ABB RAPID module: PointDesignationR.mod

MODULE PointDesignationR

    CONST robtarget CameraHome:=[[337.1108,-127.6151,556.8743],[0.2459916,-0.1669462,-0.7414577,-0.601546],[1,0,1,4],[-163.8462,9E+09,9E+09,9E+09,9E+09,9E+09]];
    CONST robtarget CameraCapture:=[[239.1137,358.6136,539.5127],[0.0857302,0.05589002,-0.9655566,-0.2392219],[1,-1,1,0],[-145.4031,9E+09,9E+09,9E+09,9E+09,9E+09]];
    CONST robtarget start:=[[642.9492,-111.2745,468.2284],[0.1105639,0.6696309,0.7196313,0.1466322],[0,0,1,4],[114.9814,9E+09,9E+09,9E+09,9E+09,9E+09]];
    CONST robtarget p1:=[[563.1667,1.634485,471.787],[0.03260814,0.4073159,0.8776615,0.250481],[0,0,1,4],[147.4612,9E+09,9E+09,9E+09,9E+09,9E+09]];
    CONST robtarget p2:=[[460.5015,84.74587,473.8824],[0.008372958,-0.2721901,-0.9279103,-0.2546074],[0,0,1,4],[155.3859,9E+09,9E+09,9E+09,9E+09,9E+09]];

    CONST robtarget HomeTest:=[[332.0402,-329.8491,328.352],[0.4885546,-0.5209683,0.4893349,-0.5004576],[0,-3,1,4],[168.771,9E+09,9E+09,9E+09,9E+09,9E+09]];
    CONST robtarget HoToDis:=[[494.5024,-289.6072,161.4639],[0.01505137,-0.03083308,0.6936113,-0.7195319],[1,-1,1,4],[138.7453,9E+09,9E+09,9E+09,9E+09,9E+09]];
    CONST robtarget DisP:=[[482.48,-440.14,154.17],[0.00187341,-0.00189956,-0.707702,0.706506],[1,-2,1,4],[169.021,9E+09,9E+09,9E+09,9E+09,9E+09]];
    CONST robtarget DisPClose:=[[482.48,-378.29,154.17],[0.00187371,-0.00189861,-0.707701,0.706507],[1,-2,1,4],[169.021,9E+09,9E+09,9E+09,9E+09,9E+09]];
    CONST robtarget DisPAbove:=[[479.74,-441.56,285.22],[0.00187343,-0.00192305,-0.70768,0.706528],[1,-2,0,4],[169.013,9E+09,9E+09,9E+09,9E+09,9E+09]];
    CONST robtarget Noz1Above:=[[376.7062,-377.0453,343.9259],[0.0008304672,-0.002048479,-0.7044001,0.7097998],[0,-1,1,4],[134.22,9E+09,9E+09,9E+09,9E+09,9E+09]];
    CONST robtarget Noz1SLAbove:=[[376.7062,-377.0453,300.9713],[0.0008473364,-0.00203507,-0.7044098,0.7097901],[0,-1,1,4],[134.2202,9E+09,9E+09,9E+09,9E+09,9E+09]];
    CONST robtarget Noz1:=[[376.7062,-377.0453,279.41],[0.000817602,-0.00204644,-0.704387,0.709812],[0,-1,1,4],[134.215,9E+09,9E+09,9E+09,9E+09,9E+09]];
    CONST robtarget NozHome:=[[423.2646,-445.0486,381.9582],[0.001873649,-0.00192683,-0.7076838,0.7065242],[0,-2,0,4],[169.0306,9E+09,9E+09,9E+09,9E+09,9E+09]];
    CONST robtarget Pos_1:=[[434.8479,154.5885,276.2301],[0.2389856,-0.6773704,0.6690471,-0.1908697],[0,-1,0,0],[137.3644,9E+09,9E+09,9E+09,9E+09,9E+09]];
    CONST robtarget Pos_2:=[[508.7112,154.7467,276.2278],[0.2344545,-0.6661509,0.682647,-0.1877956],[0,-1,0,0],[137.3715,9E+09,9E+09,9E+09,9E+09,9E+09]];
    CONST robtarget Pos_3:=[[445.0982,69.16022,245.3284],[0.2387831,-0.6774528,0.6691095,-0.1906116],[2,-1,0,0],[129.9543,9E+09,9E+09,9E+09,9E+09,9E+09]];
    CONST robtarget Pos_4:=[[516.8707,70.48975,247.9003],[0.2388017,-0.6774072,0.6691476,-0.1906166],[1,-1,0,0],[130.6205,9E+09,9E+09,9E+09,9E+09,9E+09]];

    ! Camera Position for "Jars Detection" task ______ Second Approach which uses four 20 images.
    CONST robtarget Jar_1:=[[578.2363,7.590059,160.1349],[0.00247561,-0.002194457,-0.9999697,0.007042186],[1,-1,1,4],[150.582,9E+09,9E+09,9E+09,9E+09,9E+09]];
    CONST robtarget Jar_2:=[[539.0679,6.224404,160.1209],[0.002502124,-0.002170651,-0.9999694,0.007081738],[1,-1,1,4],[150.5774,9E+09,9E+09,9E+09,9E+09,9E+09]];
    CONST robtarget Jar_3:=[[506.3916,5.240112,160.1278],[0.002490915,-0.002187095,-0.9999695,0.007065233],[1,-1,1,4],[150.5787,9E+09,9E+09,9E+09,9E+09,9E+09]];
    CONST robtarget Jar_4:=[[468.2724,2.693415,160.1224],[0.002499672,-0.002171816,-0.9999694,0.007090984],[1,-1,1,4],[150.5718,9E+09,9E+09,9E+09,9E+09,9E+09]];

    CONST robtarget Jar_5:=[[467.2797,41.21567,160.1208],[0.002500687,-0.002172773,-0.9999694,0.007089187],[1,-1,1,4],[150.5729,9E+09,9E+09,9E+09,9E+09,9E+09]];
    CONST robtarget Jar_6:=[[506.2797,41.21567,160.1208],[0.002500687,-0.002172773,-0.9999694,0.007089187],[1,-1,1,4],[150.5729,9E+09,9E+09,9E+09,9E+09,9E+09]];
    CONST robtarget Jar_7:=[[539.9217,41.20918,160.1126],[0.002508863,-0.002156894,-0.9999692,0.007110072],[1,-1,1,4],[150.5725,9E+09,9E+09,9E+09,9E+09,9E+09]];
    CONST robtarget Jar_8:=[[576.3671,42.17863,160.1143],[0.002505445,-0.002157182,-0.9999692,0.007107901],[2,-1,1,4],[150.5726,9E+09,9E+09,9E+09,9E+09,9E+09]];

    CONST robtarget Jar_9:=[[575.3677,80.37881,160.1074],[0.002512477,-0.002141175,-0.9999691,0.007129352],[2,-1,1,4],[150.5705,9E+09,9E+09,9E+09,9E+09,9E+09]];
    CONST robtarget Jar_10:=[[537.2748,79.86346,160.1057],[0.002512157,-0.002139989,-0.9999691,0.007129905],[2,-1,1,4],[150.5698,9E+09,9E+09,9E+09,9E+09,9E+09]];
    CONST robtarget Jar_11:=[[502.0086,79.85998,160.1044],[0.002512725,-0.002138408,-0.9999691,0.007133875],[2,-1,1,4],[150.5689,9E+09,9E+09,9E+09,9E+09,9E+09]];
    CONST robtarget Jar_12:=[[465.7693,79.86839,160.1122],[0.002507596,-0.002156454,-0.9999692,0.007112307],[1,-1,1,4],[150.5707,9E+09,9E+09,9E+09,9E+09,9E+09]];

    CONST robtarget Jar_13:=[[465.7563,116.1511,160.1053],[0.002510817,-0.002138373,-0.9999691,0.007132343],[2,-1,1,4],[150.5686,9E+09,9E+09,9E+09,9E+09,9E+09]];
    CONST robtarget Jar_14:=[[503.1006,115.7448,160.1056],[0.0025115,-0.002136815,-0.9999691,0.007130477],[2,-1,1,4],[150.5686,9E+09,9E+09,9E+09,9E+09,9E+09]];
    CONST robtarget Jar_15:=[[538.757,114.4573,160.1061],[0.002512425,-0.002140413,-0.9999691,0.007129679],[2,-1,1,4],[150.5667,9E+09,9E+09,9E+09,9E+09,9E+09]];
    CONST robtarget Jar_16:=[[575.1255,119.2972,160.1087],[0.002503666,-0.002141883,-0.9999692,0.00712968],[2,-1,1,4],[172.0746,9E+09,9E+09,9E+09,9E+09,9E+09]];

    CONST robtarget Jar_17:=[[575.1255,155.2972,160.1087],[0.002503666,-0.002141883,-0.9999692,0.00712968],[2,-1,1,4],[172.0746,9E+09,9E+09,9E+09,9E+09,9E+09]];
    CONST robtarget Jar_18:=[[535.7615,155.2903,160.1051],[0.002497926,-0.002126256,-0.9999691,0.007146096],[2,-1,1,4],[172.0736,9E+09,9E+09,9E+09,9E+09,9E+09]];
    CONST robtarget Jar_19:=[[500.0606,153.9737,160.1045],[0.002496237,-0.002126232,-0.9999691,0.00714566],[2,-1,1,4],[172.0735,9E+09,9E+09,9E+09,9E+09,9E+09]];
    CONST robtarget Jar_20:=[[464.1317,153.2113,160.1024],[0.002497274,-0.002126625,-0.9999691,0.007149545],[2,-1,1,4],[172.0739,9E+09,9E+09,9E+09,9E+09,9E+09]];
    CONST robtarget Middle:=[[554.137,62.09487,240.156],[0.01853917,0.02127909,-0.9995263,0.01227708],[1,-1,1,4],[166.9007,9E+09,9E+09,9E+09,9E+09,9E+09]];
     ! Camera Position for "Jars Detection" task ______ First Approach which uses four images.
    VAR   robtarget Temp := [[464.1317,153.2113,160.1024],[0.002497274,-0.002126625,-0.9999691,0.007149545],[2,-1,1,4],[172.0739,9E+09,9E+09,9E+09,9E+09,9E+09]];

    CONST robtarget G{20} := [Jar_1, Jar_2, Jar_3, Jar_4, Jar_5, Jar_6, Jar_7, Jar_8, Jar_9, Jar_10, Jar_11, Jar_12, Jar_13, Jar_14, Jar_15,
        Jar_16, Jar_17, Jar_18, Jar_19, Jar_20];
    VAR num JarOnPlace{20} := [0, 0, 0, 0, 0, 0, 0, 0, 0, 0, 0, 0, 0, 0, 0, 0, 0, 0, 0, 0];
    CONST robtarget JarInPosition:=[[557.7031,199.0231,276.2335],[0.2389639,-0.6773693,0.6690513,-0.1908857],[0,-1,0,0],[137.3665,9E+09,9E+09,9E+09,9E+09,9E+09]];
    CONST robtarget JarNotInPosition:=[[557.7601,86.44871,276.2976],[0.2389937,-0.6772945,0.6690975,-0.1909521],[1,-1,0,0],[136.7944,9E+09,9E+09,9E+09,9E+09,9E+09]];

    !Nozzle positions
    VAR robtarget FirstOneOriginal:=[[364.5634,-484.9848,317.05],[0.5102121,-0.5058356,0.4925829,-0.4910968],[0,1,1,4],[146.1654,9E+09,9E+09,9E+09,9E+09,9E+09]];
    !VAR robtarget FirstOneOriginal:=[[356.2589,-488.2664,316.8112],[0.5258595,-0.4958052,0.4774238,-0.4997154],[0,-3,1,4],[-175.2839,9E+09,9E+09,9E+09,9E+09,9E+09]];
    !VAR robtarget FirstOneOriginal:=[[356.2531,-488.2716,316.8204],[0.5258421,-0.4958193,0.4774157,-0.4997275],[0,-3,1,4],[151.4595,9E+09,9E+09,9E+09,9E+09,9E+09]];
    !VAR robtarget FirstOneOriginal:=[[366.4796,-487.7165,320.9377],[0.4915279,-0.5023509,0.505054,-0.5009635],[0,1,1,4],[130.2164,9E+09,9E+09,9E+09,9E+09,9E+09]];
    VAR robtarget FirstOne:=[[356.2531,-488.2716,316.8204],[0.5258421,-0.4958193,0.4774157,-0.4997275],[0,-3,1,4],[151.4595,9E+09,9E+09,9E+09,9E+09,9E+09]];
    VAR robtarget FirstOne_20:=[[346.0473,-426.0112,432.1689],[0.5101828,-0.5058254,0.4925885,-0.4911321],[0,1,1,4],[141.0746,9E+09,9E+09,9E+09,9E+09,9E+09]];
    VAR robtarget FirstOne_21:=[[346.0473,-426.0112,432.1689],[0.5101828,-0.5058254,0.4925885,-0.4911321],[0,1,1,4],[141.0746,9E+09,9E+09,9E+09,9E+09,9E+09]];
    VAR robtarget FirstOne_13:=[[366.0591,-446.0087,432.179],[0.5101995,-0.5058179,0.4925985,-0.4911124],[0,1,1,4],[133.7709,9E+09,9E+09,9E+09,9E+09,9E+09]];
    VAR robtarget FirstOne_14:=[[346.0348,-446.0507,431.6447],[0.5101639,-0.505727,0.4926802,-0.4911611],[0,1,1,4],[148.105,9E+09,9E+09,9E+09,9E+09,9E+09]];
    VAR robtarget FirstOne_19:=[[366.0581,-426.0146,433.7001],[0.5101944,-0.5057982,0.4926129,-0.4911236],[0,1,1,4],[137.0026,9E+09,9E+09,9E+09,9E+09,9E+09]];
    VAR robtarget FirstOne_18:=[[266.2643,-445.9307,464.5445],[0.5104685,-0.5057837,0.4925609,-0.4909059],[0,1,1,4],[-118.3564,9E+09,9E+09,9E+09,9E+09,9E+09]];
    VAR robtarget FirstOne_5:=[[284.8518,-485.0245,436.239],[0.5115612,-0.5047849,0.4925893,-0.4907679],[0,1,1,4],[162.2127,9E+09,9E+09,9E+09,9E+09,9E+09]];
    VAR robtarget FirstOne_11:=[[285.39,-464.6693,439.2722],[0.5165449,-0.5008299,0.4851822,-0.4969396],[0,1,1,4],[168.0746,9E+09,9E+09,9E+09,9E+09,9E+09]];
    !opening jar lid with the right hand
    !VAR robtarget OpenJarLid_right1:=[[436.7945,-71.18093,415.3521],[0.003124756,0.7087327,0.705469,0.001334163],[0,-1,2,4],[166.2375,9E+09,9E+09,9E+09,9E+09,9E+09]];
    VAR robtarget OpenJarLid_right1:=[[436.7945,-71.18093,415.3521],[0.003124756,0.7087327,0.705469,0.001334163],[0,-1,2,4],[166.2375,9E+09,9E+09,9E+09,9E+09,9E+09]];
    VAR robtarget OpenJarLid_right1temp:=[[436.7945,-71.18093,422.3521],[0.003124756,0.7087327,0.705469,0.001334163],[0,-1,2,4],[166.2375,9E+09,9E+09,9E+09,9E+09,9E+09]];
    VAR robtarget temppp:=[[436.7945,-71.18093,421.3521],[0.003124756,0.7087327,0.705469,0.001334163],[0,-1,2,4],[166.2375,9E+09,9E+09,9E+09,9E+09,9E+09]];
    VAR jointtarget OpenJarLid_right2 := [[33.0738,-40.319,34.7805,-60.3478,90.4867,85.3075],[3.62614,9E+09,9E+09,9E+09,9E+09,9E+09]];
    VAR jointtarget OpenJarLid_right3 := [[33.0794,-39.967,34.5252,-60.3689,90.4027,14.3972],[3.62142,9E+09,9E+09,9E+09,9E+09,9E+09]];
    !points for TakeOutJarLidAndCloseJar
    VAR robtarget TakeOutJarLidAndCloseJar1:=[[548.4954,-84.25315,36.47867],[0.001396735,-0.7047526,-0.7094415,0.003806988],[1,-1,2,4],[152.5241,9E+09,9E+09,9E+09,9E+09,9E+09]];
    VAR robtarget TakeOutJarLidAndCloseJar1Temp:=[[548.4954,-84.25315,36.47867],[0.001396735,-0.7047526,-0.7094415,0.003806988],[1,-1,2,4],[152.5241,9E+09,9E+09,9E+09,9E+09,9E+09]];
    VAR robtarget TakeOutJarLidAndCloseJar2:=[[549.129,-86.93868,70.51934],[0.005022825,0.7009446,0.7131749,-0.005741474],[1,-1,2,4],[148.9269,9E+09,9E+09,9E+09,9E+09,9E+09]];
    VAR robtarget TakeOutJarLidAndCloseJar3:=[[530.686,-275.6855,198.1201],[0.005085662,0.7029518,0.7111219,0.01177542],[0,-1,1,4],[144.7235,9E+09,9E+09,9E+09,9E+09,9E+09]];
    VAR robtarget TakeOutJarLidAndCloseJar4:=[[442.0807,-71.82523,457.5505],[0.004448493,-0.7243365,-0.6894255,-0.003039069],[0,-1,2,4],[175.2385,9E+09,9E+09,9E+09,9E+09,9E+09]];
    VAR robtarget TakeOutJarLidAndCloseJar5:=[[544.5369,-219.8828,495.8261],[0.03485789,0.6806227,0.731776,0.00644785],[0,-1,1,4],[165.815,9E+09,9E+09,9E+09,9E+09,9E+09]];
    !points for closing jar lid
    VAR robtarget CloseJarLid_right1:=[[436.7945,-71.18093,415.3521],[0.003124756,0.7087327,0.705469,0.001334163],[0,-1,2,4],[166.2375,9E+09,9E+09,9E+09,9E+09,9E+09]];
    VAR jointtarget CloseJarLid_right2 := [[33.0738,-40.319,34.7805,-60.3478,90.4867,85.3075],[3.62614,9E+09,9E+09,9E+09,9E+09,9E+09]];
    VAR jointtarget CloseJarLid_right3 := [[33.0738,-40.319,34.7805,-60.3478,90.4867,85.3075],[3.62614,9E+09,9E+09,9E+09,9E+09,9E+09]];

    ! Some points to calibrate the lid on the yellow station.
    VAR robtarget Calibration_1 := [[580.5686,-88.29684,34.52171],[0.001399272,-0.7047435,-0.7094505,0.003823198],[1,-1,1,4],[152.5257,9E+09,9E+09,9E+09,9E+09,9E+09]];
    VAR robtarget Calibration_2 := [[565.8522,-88.29948,34.51547],[0.001400438,-0.7047327,-0.7094612,0.003840852],[1,-1,1,4],[152.5268,9E+09,9E+09,9E+09,9E+09,9E+09]];
    VAR robtarget Calibration_3 := [[580.5543,-88.29913,63.13507],[0.001398228,-0.7047324,-0.7094615,0.003841279],[1,-1,1,4],[152.5264,9E+09,9E+09,9E+09,9E+09,9E+09]];

    ! Points to Pick the Pippete by the right arm
    VAR robtarget PickPippete1 := [[195.649,-319.5563,313.2436],[0.7112405,-0.6988382,-0.01608902,0.07418307],[0,0,1,4],[149.918,9E+09,9E+09,9E+09,9E+09,9E+09]];
    VAR robtarget PickPippete2 := [[170.5461,-230.7654,213.2043],[0.7046992,-0.7058032,-0.01402912,0.07102092],[0,0,1,4],[157.0625,9E+09,9E+09,9E+09,9E+09,9E+09]];
    VAR robtarget PickPippete3 := [[175.5379,-131.7484,179.4989],[0.7079524,-0.7062595,0.000795693,-0.0004416163],[1,0,1,4],[156.2807,9E+09,9E+09,9E+09,9E+09,9E+09]];
    VAR robtarget PickPippeteNearPippete := [[177.2253,-197.436,179.0786],[0.7079537,-0.7062583,0.0007935975,-0.0004423254],[1,0,1,4],[156.2809,9E+09,9E+09,9E+09,9E+09,9E+09]];
    VAR robtarget PickPippeteAroundPippete := [[177.222,-131.1301,179.0808],[0.7079551,-0.7062569,0.0007965097,-0.0004404763],[1,0,1,4],[156.2794,9E+09,9E+09,9E+09,9E+09,9E+09]];
    VAR robtarget PickPippeteAroundPippeteTemp := [[175.5381,-135.7663,177.2376],[0.7079375,-0.7062744,0.0007983644,-0.0004442568],[1,0,1,4],[156.2761,9E+09,9E+09,9E+09,9E+09,9E+09]];
    VAR robtarget PickPippete4 := [[175.5398,-131.7487,239.373],[0.7079531,-0.7062589,0.0007958095,-0.0004424199],[0,0,1,4],[156.2839,9E+09,9E+09,9E+09,9E+09,9E+09]];
    VAR robtarget PickPippete9 := [[58.00851,-512.0497,345.0829],[0.4806274,-0.1937006,-0.4309853,0.7387348],[0,-1,1,4],[143.3251,9E+09,9E+09,9E+09,9E+09,9E+09]];

    VAR robtarget PickPippete4_1 := [[175.5398,-131.7487,239.373],[0.7079531,-0.7062589,0.0007958095,-0.0004424199],[0,0,1,4],[156.2839,9E+09,9E+09,9E+09,9E+09,9E+09]];
    VAR robtarget PickPippete4_2 := [[177.189,-129.7891,184.7826],[0.7079679,-0.7062441,0.0007926978,-0.0004394072],[1,0,1,4],[156.297,9E+09,9E+09,9E+09,9E+09,9E+09]];
    VAR robtarget PickPippete4_3 := [[177.1892,-131.3987,179.9682],[0.7079687,-0.7062433,0.0007927868,-0.0004407596],[1,0,1,4],[156.2953,9E+09,9E+09,9E+09,9E+09,9E+09]];
    VAR robtarget PickPippete5 := [[175.54,-84.27259,239.3745],[0.7079518,-0.7062601,0.0007943012,-0.0004460925],[0,0,1,4],[156.2846,9E+09,9E+09,9E+09,9E+09,9E+09]];
    VAR robtarget PickPippete6 := [[210.1792,-67.51133,340.1431],[0.707966,-0.7062459,0.000791344,-0.0005087436],[0,0,1,4],[156.2923,9E+09,9E+09,9E+09,9E+09,9E+09]];
    VAR robtarget PickPippete7 := [[210.188,-262.3564,340.1374],[0.7079696,-0.7062423,0.0007848368,-0.0005118064],[0,0,1,4],[156.2934,9E+09,9E+09,9E+09,9E+09,9E+09]];
    VAR robtarget PickPippete8 := [[125.4009,-534.7796,414.5038],[0.131219,-0.2493133,-0.5331899,0.7977049],[0,-2,1,4],[151.5354,9E+09,9E+09,9E+09,9E+09,9E+09]];
    !VAR robtarget PickPippete9 := [[210.188,-262.3564,340.1374],[0.7079696,-0.7062423,0.0007848368,-0.0005118064],[0,0,1,4],[156.2934,9E+09,9E+09,9E+09,9E+09,9E+09]];

    ! Points to fill in thpippetee pippete:
    VAR robtarget FillPippete1 := [[341.6258,-683.9443,511.5084],[0.3637904,0.08358209,0.7211897,-0.5835717],[0,-2,1,4],[124.8139,9E+09,9E+09,9E+09,9E+09,9E+09]];
    VAR robtarget FillPippete2 := [[62.87461,-589.7764,515.0416],[0.275436,-0.4339039,-0.530328,0.6742511],[0,-1,1,4],[83.96245,9E+09,9E+09,9E+09,9E+09,9E+09]];
    VAR robtarget FillPippete3 := [[94.98569,-349.8907,431.9817],[0.5727671,-0.7467703,-0.2549731,0.2219474],[0,0,1,4],[102.5853,9E+09,9E+09,9E+09,9E+09,9E+09]];
    VAR robtarget FillPippete4 := [[325.1082,-268.9037,457.7535],[0.6786064,-0.7311609,0.02967721,-0.06337433],[0,0,1,4],[119.312,9E+09,9E+09,9E+09,9E+09,9E+09]];
    VAR robtarget FillPippete5 := [[518.0054,-173.6114,458.7383],[0.6916274,-0.7042932,0.08632144,-0.1348009],[0,0,2,4],[141.7079,9E+09,9E+09,9E+09,9E+09,9E+09]];
    VAR robtarget FillPippete5_2 := [[325.9447,-448.3383,517.3318],[0.500117,-0.5342081,0.4917862,-0.4718592],[0,1,2,4],[19.87668,9E+09,9E+09,9E+09,9E+09,9E+09]];
    VAR robtarget FillPippete6 := [[406.7556,-112.5167,413.2942],[0.7238337,-0.6896673,-0.02013941,-0.004262863],[0,1,1,4],[111.738,9E+09,9E+09,9E+09,9E+09,9E+09]];
    VAR robtarget FillPippeteAbovePillar := [[382.0186,-119.6331,401.914],[0.7184521,-0.6954185,0.002709595,0.01457028],[0,1,1,4],[107.1083,9E+09,9E+09,9E+09,9E+09,9E+09]];
    VAR robtarget FillPippeteOnPillar := [[379.1049,-119.6783,294.4594],[0.7053983,-0.7086881,-0.009383416,0.009290063],[0,1,1,4],[109.6973,9E+09,9E+09,9E+09,9E+09,9E+09]];

    ! Points to fill out the pippetee pippete:
    VAR robtarget EmptyPippete1 := [[194.0893,-78.50488,327.2501],[0.7140521,-0.7000166,0.009698046,0.003494652],[0,0,2,4],[-157.3246,9E+09,9E+09,9E+09,9E+09,9E+09]];
    VAR robtarget EmptyPippete2 := [[210.188,-262.3564,340.1374],[0.7079696,-0.7062423,0.0007848368,-0.0005118064],[0,0,1,4],[156.2934,9E+09,9E+09,9E+09,9E+09,9E+09]];
    VAR robtarget EmptyPippeteAbovePillar := [[305.8019,-119.6324,415.2216],[0.7184599,-0.6954104,0.002705107,0.01457578],[0,0,1,4],[107.1128,9E+09,9E+09,9E+09,9E+09,9E+09]];
    VAR robtarget EmptyPippeteOnPillar := [[305.8099,-129.6291,343.5904],[0.7184706,-0.6953998,0.002716619,0.01455591],[0,0,1,4],[107.1226,9E+09,9E+09,9E+09,9E+09,9E+09]];

    ! points for the process "MovToDropNozzel"
    VAR robtarget MovToDropNozzel_1 := [[226.4902,-77.93933,422.6241],[0.7088562,-0.7053393,-0.002122149,-0.003846428],[0,0,2,4],[169.3425,9E+09,9E+09,9E+09,9E+09,9E+09]];
    VAR robtarget MovToDropNozzel_2 := [[214.2217,-84.88783,308.7547],[0.7059045,-0.7081568,-0.002914121,0.01429262],[0,0,2,4],[-162.09,9E+09,9E+09,9E+09,9E+09,9E+09]];
    VAR robtarget MovToDropNozzel_3 := [[235.3263,-130.4883,301.9571],[0.7004695,-0.698977,-0.09645084,0.1071022],[0,0,2,4],[-165.3392,9E+09,9E+09,9E+09,9E+09,9E+09]];
    VAR robtarget MovToDropNozzel_4 := [[238.051,-129.9063,296.7406],[0.7143627,-0.6905517,-0.07245048,0.08703598],[0,0,2,4],[-164.1591,9E+09,9E+09,9E+09,9E+09,9E+09]];

    VAR robtarget MovToDropNozzel_11 := [[255.6884,-123.6689,417.4043],[0.7184788,-0.6953905,0.002693033,0.0145991],[0,0,1,4],[107.1369,9E+09,9E+09,9E+09,9E+09,9E+09]];
    VAR robtarget MovToDropNozzel_22 := [[260.9324,-133.7218,343.3578],[0.7184805,-0.6953891,0.002707851,0.01457953],[0,0,1,4],[107.1803,9E+09,9E+09,9E+09,9E+09,9E+09]];


    !points to open held jar
    VAR robtarget Midd1:=[[516.37,-146.3473,438.789],[0.130924,-0.6841183,-0.6827902,-0.2205418],[0,0,1,4],[155.2096,9E+09,9E+09,9E+09,9E+09,9E+09]];
    VAR robtarget Midd2:=[[548.4106,-86.3063,203.8174],[0.03204845,0.7046776,0.7087683,-0.007059979],[0,-1,2,4],[126.0521,9E+09,9E+09,9E+09,9E+09,9E+09]];
    VAR robtarget Midd9:=[[533.0876,-139.4853,36.35339],[0.3614811,-0.9298749,-0.06503172,-0.02085684],[1,0,2,4],[148.8922,9E+09,9E+09,9E+09,9E+09,9E+09]];
    VAR robtarget Midd10:=[[555.2894,-147.5639,78.93652],[0.4163733,-0.9058304,-0.07784346,-0.006713092],[1,0,2,4],[147.3773,9E+09,9E+09,9E+09,9E+09,9E+09]];
    VAR robtarget Midd11:=[[552.0694,-185.2786,192.0681],[0.2910097,-0.9447768,-0.150038,-0.01409988],[1,0,2,4],[136.7552,9E+09,9E+09,9E+09,9E+09,9E+09]];
    VAR robtarget Midd12:=[[376.4778,-621.3032,351.6772],[0.2155167,0.121452,0.6633735,-0.7062135],[0,-2,1,4],[137.6339,9E+09,9E+09,9E+09,9E+09,9E+09]];
    VAR robtarget Midd13:=[[405.1425,-425.9179,278.2724],[0.06600403,-0.6850826,-0.6951225,0.2076298],[0,-1,1,4],[138.5983,9E+09,9E+09,9E+09,9E+09,9E+09]];
    VAR robtarget Midd14:=[[524.7402,-220.1512,231.3111],[0.08746707,-0.7491345,-0.6542986,-0.0551387],[0,0,1,4],[126.5334,9E+09,9E+09,9E+09,9E+09,9E+09]];
    VAR robtarget Midd15:=[[547.8265,-140.1339,118.4852],[0.001163659,-0.7173198,-0.6967209,0.005557916],[0,0,1,0],[106.4498,9E+09,9E+09,9E+09,9E+09,9E+09]];
    VAR robtarget Midd16:=[[537.3522,-140.5765,56.02523],[0.0006988946,0.7074742,0.706738,-0.001055677],[0,0,1,0],[95.53145,9E+09,9E+09,9E+09,9E+09,9E+09]];
    VAR robtarget Midd17:=[[537.3522,-140.5782,35.26651],[0.0006965169,0.7074735,0.7067387,-0.001056443],[0,0,1,0],[95.53266,9E+09,9E+09,9E+09,9E+09,9E+09]];
    VAR robtarget Midd18:=[[528.0477,-182.1228,174.811],[0.0147931,-0.7378669,-0.6738108,-0.0362289],[0,0,1,4],[110.359,9E+09,9E+09,9E+09,9E+09,9E+09]];
    VAR robtarget Midd19:=[[540.8347,-79.36512,185.1231],[0.02389621,0.6877341,0.7253837,-0.01640796],[0,-1,1,0],[121.6245,9E+09,9E+09,9E+09,9E+09,9E+09]];

    VAR robtarget Midd20:=[[524.5283,-396.8792,239.3516],[0.01855994,0.6776902,0.7351087,-0.002606999],[0,-1,1,4],[129.2266,9E+09,9E+09,9E+09,9E+09,9E+09]];
    VAR robtarget Midd21:=[[548.7518,-434.0228,175.894],[0.1244405,0.6483645,0.7493331,-0.05136107],[1,-1,1,4],[135.195,9E+09,9E+09,9E+09,9E+09,9E+09]];
    VAR robtarget Midd22:=[[519.0132,-376.5699,295.0557],[0.116374,-0.6922324,-0.6913291,-0.1712761],[0,-1,1,4],[158.3923,9E+09,9E+09,9E+09,9E+09,9E+09]];
    VAR robtarget Midd23:=[[632.9103,-23.5132,150.1017],[0.0006158123,0.04710628,0.9988896,0.0003107161],[1,-1,1,4],[175.2924,9E+09,9E+09,9E+09,9E+09,9E+09]];

    VAR robtarget Midd5:=[[535.7374,-133.5883,40.87439],[0.01621619,-0.7097876,-0.7039508,-0.01979489],[1,-1,1,4],[151.373,9E+09,9E+09,9E+09,9E+09,9E+09]];
    VAR robtarget Midd6:=[[528.7254,-168.0216,66.49234],[0.1161043,-0.7062157,-0.6848287,-0.1370725],[1,-1,1,4],[149.4186,9E+09,9E+09,9E+09,9E+09,9E+09]];
    VAR robtarget Midd7:=[[535.4856,-138.1096,66.77904],[0.3913096,-0.9191372,-0.02135808,-0.04009253],[1,0,1,4],[141.1107,9E+09,9E+09,9E+09,9E+09,9E+09]];
    VAR robtarget Midd8:=[[540.0371,-122.9395,36.96175],[0.3743683,-0.9270967,-0.01667459,0.007885762],[1,0,2,4],[148.7738,9E+09,9E+09,9E+09,9E+09,9E+09]];
    VAR robtarget HeldJar_PickCover:=[[550.4392,-88.55307,35.23132],[0.0004738881,-0.711928,-0.7022521,-0.0004824866],[1,-1,2,4],[151.1626,9E+09,9E+09,9E+09,9E+09,9E+09]];
    VAR robtarget HeldJar_PickCoverTemp:=[[550.8508,-90.06332,34.75971],[0.01568587,-0.7116391,-0.702301,0.009851178],[1,-1,2,4],[151.1403,9E+09,9E+09,9E+09,9E+09,9E+09]];
    VAR robtarget Midd3:=[[536.4565,-105.2238,209.9932],[0.0009176944,-0.6966414,-0.7165335,-0.03563081],[0,-1,1,4],[131.0546,9E+09,9E+09,9E+09,9E+09,9E+09]];
    VAR robtarget HeldJar_AboveJar:=[[541.1,-80.88705,166.6814],[0.01086609,0.6972497,0.7166983,-0.008257998],[0,0,1,0],[113.2381,9E+09,9E+09,9E+09,9E+09,9E+09]];
    VAR robtarget HeldJar_PlaceCover:=[[541.0815,-80.86801,150.2539],[0.01083725,0.6972349,0.716713,-0.008280328],[0,-1,1,0],[113.2341,9E+09,9E+09,9E+09,9E+09,9E+09]];
    VAR robtarget HeldJar_PlaceCover2:=[[467.9971,59.64725,138.2034],[0.0001647275,0.3948865,0.9187299,1.392494E-05],[1,-1,1,4],[155.6173,9E+09,9E+09,9E+09,9E+09,9E+09]];
    VAR robtarget Midd4:=[[545.335,-169.6051,166.0662],[0.007297219,0.6852906,0.7281541,-0.01073433],[1,-1,1,4],[138.3401,9E+09,9E+09,9E+09,9E+09,9E+09]];
    VAR jointtarget OpenHeldJarLid_right2 := [[122.646,-32.5409,13.8014,-101.023,71.2433,154.106],[-109.167,9E+09,9E+09,9E+09,9E+09,9E+09]];
    VAR robtarget Held_OpenJarLid_right1:=[[299.925,-104.7758,141.8612],[0.003347919,0.5523319,-0.8336176,-0.0001573839],[1,-1,0,4],[177.4993,9E+09,9E+09,9E+09,9E+09,9E+09]];
    VAR robtarget Held_OpenJarLid_right3 := [[466.0024,63.63331,142.2465],[0.0001546609,0.5512216,0.8343589,6.732765E-05],[1,-1,2,4],[155.6186,9E+09,9E+09,9E+09,9E+09,9E+09]];
    VAR robtarget Held_OpenJarLid_right1_Orig:=[[464.5274,59.26692,140.2369],[0.0001036231,-0.5265943,0.8501167,-0.0001247879],[1,-1,0,4],[155.6124,9E+09,9E+09,9E+09,9E+09,9E+09]];
    VAR robtarget Held_OpenJarLid_right3_Orig := [[466.1872,57.94262,140.2382],[0.000161748,0.5219612,0.8529692,3.900014E-05],[1,-1,2,4],[155.612,9E+09,9E+09,9E+09,9E+09,9E+09]];
    VAR robtarget Held_OpenJarLid_right11_Orig:=[[540.0129,-79.90893,145.1838],[0.0009086653,-0.04636181,0.9989234,0.001365947],[0,0,0,0],[105.7546,9E+09,9E+09,9E+09,9E+09,9E+09]];
    VAR robtarget Held_OpenJarLid_right33_Orig := [[540.1237,-80.10228,145.1842],[0.0008563087,-0.8882292,-0.4593977,-0.001396758],[0,0,2,0],[105.7547,9E+09,9E+09,9E+09,9E+09,9E+09]];
    VAR robtarget Held_OpenJarLid_right2 := [[467.3242,60.99391,142.2465],[0.0001546609,0.5512216,0.8343589,6.732765E-05],[1,-1,2,4],[155.6186,9E+09,9E+09,9E+09,9E+09,9E+09]];
    VAR jointtarget HeldJar_PlaceCoverAbs := [[119.341,-29.4085,15.7471,-99.831,65.08,129.757],[-107.428,9E+09,9E+09,9E+09,9E+09,9E+09]];
    VAR robtarget Held_PushingCover:=[[467.1174,60.89045,139.2775],[0.0001697346,0.1287424,0.9916781,1.377234E-05],[1,-1,1,4],[155.6257,9E+09,9E+09,9E+09,9E+09,9E+09]];
    VAR robtarget PushingPoint:=[[466.9691,60.80544,139.272],[0.0001234702,-0.5892357,0.8079612,-0.0001076188],[1,-1,0,4],[155.6251,9E+09,9E+09,9E+09,9E+09,9E+09]];

    VAR jointtarget Held_PushingCoverABS := [[122.099,-29.6605,14.5162,-99.2677,66.8305,97.9901],[-109.49,9E+09,9E+09,9E+09,9E+09,9E+09]];

    VAR robtarget Held_RightRest:=[[580.5162,-291.4563,179.9309],[0.007601542,0.7500571,0.6528434,0.1056029],[1,0,1,4],[123.5707,9E+09,9E+09,9E+09,9E+09,9E+09]];
    VAR jointtarget PushingPointABS := [[122.106,-29.6623,14.5238,-99.2724,66.8321,129.732],[-109.493,9E+09,9E+09,9E+09,9E+09,9E+09]];
    !Points to pick new filter
    VAR robtarget PickNewFilter1 := [[621.5493,-320.5108,393.9513],[0.7063952,-0.1006195,0.6996402,0.03721725],[0,1,2,4],[126.3033,9E+09,9E+09,9E+09,9E+09,9E+09]];
    VAR robtarget InsideFiltersContainer1 := [[624.0345,-425.5425,83.53399],[0.6080498,0.2930888,0.6843289,-0.2758049],[1,2,2,4],[-179.9588,9E+09,9E+09,9E+09,9E+09,9E+09]];
    VAR robtarget InsideFiltersContainer2 := [[627.1578,-426.0681,114.7737],[0.6080431,0.2930834,0.6843358,-0.2758084],[1,2,1,4],[-179.9476,9E+09,9E+09,9E+09,9E+09,9E+09]];
    VAR robtarget InsideFiltersContainer3 := [[627.1589,-424.3743,83.64411],[0.6080429,0.2930817,0.6843359,-0.2758102],[1,2,2,4],[-179.9422,9E+09,9E+09,9E+09,9E+09,9E+09]];
    VAR robtarget PickNewFilter3 := [[700.8572,-123.4617,503.5828],[0.6779857,-0.2063949,0.6670991,0.2295984],[0,1,2,4],[148.6769,9E+09,9E+09,9E+09,9E+09,9E+09]];
    VAR robtarget PlaceFilterOnBigJar := [[748.2884,-71.93338,425.3625],[0.7177004,-0.2530347,0.6101761,0.2203737],[1,1,2,4],[161.6583,9E+09,9E+09,9E+09,9E+09,9E+09]];
!    VAR robtarget PlaceFilterOnBigJar := [[746.3795,-64.11948,423.8503],[0.6907627,-0.2801198,0.6255661,0.230319],[1,1,2,4],[159.9187,9E+09,9E+09,9E+09,9E+09,9E+09]];
    VAR robtarget FilterAboveBigJar := [[736.3964,-58.74627,465.7315],[0.7179585,-0.3043995,0.571655,0.255122],[1,1,2,4],[164.984,9E+09,9E+09,9E+09,9E+09,9E+09]];
    VAR robtarget AboveFiltersContainer1 := [[624.0604,-425.5498,98.79743],[0.6080633,0.2930799,0.6843215,-0.2758029],[1,2,2,4],[-179.9616,9E+09,9E+09,9E+09,9E+09,9E+09]];
    VAR robtarget AboveFiltersContainer1_1 := [[594.6089,-425.1374,364.7184],[0.6710457,0.227214,0.6689132,-0.2250035],[0,2,1,4],[167.9116,9E+09,9E+09,9E+09,9E+09,9E+09]];
    VAR robtarget AboveFiltersContainer2 := [[624.0294,-425.5365,91.14505],[0.6080458,0.2930862,0.6843331,-0.2758062],[1,2,2,4],[-179.9555,9E+09,9E+09,9E+09,9E+09,9E+09]];
    VAR robtarget AboveFiltersContainer3 := [[624.0205,-437.218,91.17622],[0.6080415,0.2930878,0.6843355,-0.2758076],[1,2,2,4],[-179.9546,9E+09,9E+09,9E+09,9E+09,9E+09]];
    VAR robtarget AboveFiltersContainer4 := [[627.1556,-424.3723,122.1105],[0.6080418,0.2930837,0.6843366,-0.275809],[1,2,1,4],[-179.9405,9E+09,9E+09,9E+09,9E+09,9E+09]];
    VAR robtarget PickNewFilter6 := [[496.8484,-96.40296,487.0166],[0.1605303,-0.5834689,-0.756124,-0.2491398],[0,0,1,4],[166.8297,9E+09,9E+09,9E+09,9E+09,9E+09]];
    VAR robtarget PickNewFilter7 := [[457.8124,-35.79226,579.4077],[0.3662375,-0.4543677,-0.6626154,-0.4694262],[0,0,1,4],[166.312,9E+09,9E+09,9E+09,9E+09,9E+09]];
    VAR robtarget AbovePlate := [[624.5128,-458.676,421.1502],[0.5257624,0.4944812,0.4941018,-0.4846913],[1,-2,1,4],[165.4171,9E+09,9E+09,9E+09,9E+09,9E+09]];
    VAR robtarget AbovePlate_Suck := [[634.1646,-464.1222,378.8921],[0.512431,0.4822668,0.5282508,-0.4751677],[1,-2,1,4],[164.8169,9E+09,9E+09,9E+09,9E+09,9E+09]];

    !Points to pick and place funnel
    VAR robtarget PickAndPlaceFunnel1 := [[624.5128,-458.676,421.1502],[0.5257624,0.4944812,0.4941018,-0.4846913],[1,-2,1,4],[165.4171,9E+09,9E+09,9E+09,9E+09,9E+09]];
    VAR robtarget PickAndPlaceFunnel2 := [[574.0182,-349.3656,158.0238],[0.4653983,0.4840121,0.541185,0.5062168],[1,1,-1,4],[-175.8753,9E+09,9E+09,9E+09,9E+09,9E+09]];
    VAR robtarget PickAndPlaceFunnel3 := [[680.494,-358.076,380.4701],[0.5418031,-0.5262768,0.4639729,-0.4628298],[1,1,1,4],[172.4639,9E+09,9E+09,9E+09,9E+09,9E+09]];
    VAR robtarget PickAndPlaceFunnel4 := [[658.501,-109.3655,429.152],[0.6591876,-0.669107,0.2579699,-0.2263163],[1,1,2,4],[155.3449,9E+09,9E+09,9E+09,9E+09,9E+09]];
    VAR robtarget FunnelOnBigJar := [[667.3174,-109.5582,366.937],[0.66706,-0.6810696,0.2161981,-0.2107928],[1,1,2,4],[150.1866,9E+09,9E+09,9E+09,9E+09,9E+09]];
    VAR robtarget FunnelAboveBigJar := [[662.0784,-110.5511,435.6039],[0.6728038,-0.6753909,0.2155411,-0.2114811],[1,1,2,4],[149.9029,9E+09,9E+09,9E+09,9E+09,9E+09]];
    CONST robtarget NearFunnel := [[598.678,-340.9526,110.1934],[0.5140692,0.513207,0.4848319,0.4871237],[1,1,-1,4],[-173.0962,9E+09,9E+09,9E+09,9E+09,9E+09]];
    CONST robtarget AroundFunnel := [[668.3562,-341.1264,128.9281],[0.5249498,0.5178389,0.4850127,0.4701416],[1,1,-1,4],[-163.5817,9E+09,9E+09,9E+09,9E+09,9E+09]];
    CONST robtarget AboveFunnel := [[668.3507,-341.1494,188.751],[0.5249498,0.5178389,0.4850127,0.4701416],[1,1,-1,4],[-163.5817,9E+09,9E+09,9E+09,9E+09,9E+09]];


    ! Points On The Path From Main mid-Point to Orange station, to Pick jars from JarsCarrier
!    CONST robtarget PickThenPlaceJar_1 := [[221.6189,-630.9095,263.1391],[0.1033719,-0.7078362,-0.6792379,0.1640671],[0,-1,1,4],[176.5613,9E+09,9E+09,9E+09,9E+09,9E+09]];
!    CONST robtarget PickThenPlaceJar_2 := [[182.3394,-636.3591,157.7522],[0.09313875,-0.7021877,-0.6971769,0.1104628],[0,-1,0,4],[-155.607,9E+09,9E+09,9E+09,9E+09,9E+09]];
    CONST robtarget PickThenPlaceJar_1 := [[179.2008,-636.9895,308.1646],[0.02179927,0.6937607,0.7198534,0.005655664],[0,-1,0,4],[175.8574,9E+09,9E+09,9E+09,9E+09,9E+09]];
    CONST robtarget PickThenPlaceJar_2_1 := [[178.6717,-637.1774,158.8201],[0.01474175,-0.6937976,-0.7194098,0.02961638],[0,-1,0,4],[-136.568,9E+09,9E+09,9E+09,9E+09,9E+09]];
    CONST robtarget PickThenPlaceJar_2_2 := [[178.6752,-637.1756,163.6084],[0.02207202,0.69443,0.7192031,0.005167758],[0,-1,0,4],[-136.571,9E+09,9E+09,9E+09,9E+09,9E+09]];
    CONST robtarget PickThenPlaceJar_3 := [[514.5727,-92.31973,311.4816],[0.02578642,-0.03406016,0.9988954,-0.0195672],[0,-1,1,4],[152.8023,9E+09,9E+09,9E+09,9E+09,9E+09]];
    CONST robtarget PickThenPlaceJar_4 := [[540.8358,-79.04424,241.8575],[0.01282984,-0.01291086,0.9998207,-0.005222363],[0,-1,1,4],[140.2428,9E+09,9E+09,9E+09,9E+09,9E+09]];
    CONST robtarget PickThenPlaceJar_5 := [[540.033,-79.02003,170.1638],[0.01224879,-0.01340815,0.9998229,-0.004945346],[1,-1,1,4],[140.5999,9E+09,9E+09,9E+09,9E+09,9E+09]];
    CONST robtarget PickThenPlaceJar_4_2 := [[540.827,-21.1302,241.8817],[0.01285445,-0.01293795,0.9998198,-0.005274247],[1,-1,1,4],[140.2354,9E+09,9E+09,9E+09,9E+09,9E+09]];
    CONST robtarget PickThenPlaceJar_5_2 := [[540.8089,-21.14899,197.2088],[0.01277829,-0.01288883,0.9998217,-0.005204006],[1,-1,1,4],[140.2409,9E+09,9E+09,9E+09,9E+09,9E+09]];
    CONST robtarget PickThenPlaceJar_5_3 := [[540.8538,-45.851,197.211],[0.01278042,-0.0128894,0.9998217,-0.005203976],[1,-1,1,4],[140.2329,9E+09,9E+09,9E+09,9E+09,9E+09]];


    CONST robtarget FilterFormMissileToPlate1 := [[705.6249,-118.5424,547.73],[0.7170886,-0.1016343,0.6858905,0.07077146],[1,0,-1,5],[173.9745,9E+09,9E+09,9E+09,9E+09,9E+09]];
    CONST robtarget FilterFormMissileToPlate2 := [[753.3035,-132.1059,435.7927],[0.7123696,-0.0763738,0.6961165,0.04602613],[1,0,-1,5],[171.6446,9E+09,9E+09,9E+09,9E+09,9E+09]];
    CONST robtarget FilterFormMissileToPlate3 := [[753.3035,-139.1056,418.2421],[0.7123706,-0.07637336,0.6961155,0.04602607],[1,0,-1,5],[171.6473,9E+09,9E+09,9E+09,9E+09,9E+09]];
    CONST robtarget FilterFormMissileToPlate4 := [[753.2958,-57.30429,442.5074],[0.7123702,-0.07635287,0.6961184,0.04602309],[1,0,-1,5],[171.6511,9E+09,9E+09,9E+09,9E+09,9E+09]];
    CONST robtarget FilterFormMissileToPlate5 := [[753.2941,-57.30222,411.2484],[0.7123696,-0.07635479,0.6961186,0.04602571],[1,0,-1,5],[171.6533,9E+09,9E+09,9E+09,9E+09,9E+09]];

    !Points to push filter on big jar
    VAR robtarget PushFilter1 := [[756.0059,-13.61446,394.8519],[0.02664099,-0.762088,-0.2717999,-0.5870579],[1,0,0,5],[170.9841,9E+09,9E+09,9E+09,9E+09,9E+09]];
    VAR robtarget PushFilter2 := [[756.8353,-17.41819,380.0923],[0.02663975,-0.7620836,-0.2718007,-0.5870632],[1,0,0,5],[170.9992,9E+09,9E+09,9E+09,9E+09,9E+09]];
    VAR robtarget PushFilter3 := [[749.9757,-27.72997,380.5538],[0.02663724,-0.762088,-0.2718012,-0.5870575],[1,0,1,5],[170.9892,9E+09,9E+09,9E+09,9E+09,9E+09]];
    VAR robtarget PushFilter4 := [[743.4111,-33.86438,380.5558],[0.02663806,-0.7620863,-0.2718004,-0.5870599],[1,0,1,5],[170.9918,9E+09,9E+09,9E+09,9E+09,9E+09]];
    VAR robtarget PushFilter5 := [[737.4625,-40.36673,380.5567],[0.02663708,-0.7620859,-0.2718003,-0.5870607],[1,0,1,5],[170.9944,9E+09,9E+09,9E+09,9E+09,9E+09]];
    VAR robtarget PushFilter6 := [[733.3664,-46.5193,380.5568],[0.02663536,-0.7620849,-0.2718024,-0.587061],[1,0,1,5],[170.9958,9E+09,9E+09,9E+09,9E+09,9E+09]];
    VAR robtarget PushFilter7 := [[733.374,-46.5389,389.5945],[0.02661256,-0.7620885,-0.2717963,-0.5870603],[1,0,1,5],[170.9965,9E+09,9E+09,9E+09,9E+09,9E+09]];
    VAR robtarget PushFilter8 := [[733.368,-46.54215,458.1636],[0.02660939,-0.7620866,-0.2717976,-0.5870622],[1,1,0,5],[170.9965,9E+09,9E+09,9E+09,9E+09,9E+09]];
    VAR robtarget PushFilter9 := [[741.5504,-50.15194,502.4712],[0.1524157,0.3446489,0.7166551,0.5868492],[1,0,1,4],[175.4269,9E+09,9E+09,9E+09,9E+09,9E+09]];
    VAR robtarget PushFilter10 := [[736.2281,-82.81029,382.6262],[0.5206777,-0.2948277,0.801129,-0.01278638],[1,1,2,5],[162.8944,9E+09,9E+09,9E+09,9E+09,9E+09]];
    VAR robtarget PushFilter11 := [[724.3495,-65.00657,382.1458],[0.527997,-0.3223275,0.7825246,0.0705651],[1,1,2,5],[159.5265,9E+09,9E+09,9E+09,9E+09,9E+09]];
    VAR robtarget PushFilter12 := [[728.5455,-49.11105,419.8861],[0.5490216,-0.3086144,0.7727147,0.07902226],[1,1,2,5],[161.8061,9E+09,9E+09,9E+09,9E+09,9E+09]];
    VAR robtarget PushFilter13 := [[743.5784,25.86427,430.176],[0.6582333,-0.2462072,0.6854758,0.1903519],[1,1,2,0],[121.1031,9E+09,9E+09,9E+09,9E+09,9E+09]];
    VAR robtarget PushFilter14 := [[733.2577,-46.34735,458.0763],[0.5866504,-0.3494981,0.7297264,-0.03452196],[1,1,2,5],[170.9967,9E+09,9E+09,9E+09,9E+09,9E+09]];
    VAR robtarget PushFilter15 := [[801.3381,-85.08338,551.8134],[0.510915,0.341691,0.7031891,0.3574048],[0,0,1,0],[130.876,9E+09,9E+09,9E+09,9E+09,9E+09]];
    VAR robtarget PushFilter16 := [[664.3308,-108.3452,397.178],[0.006608484,0.4401534,0.897898,0.0006642516],[0,0,1,0],[130.8481,9E+09,9E+09,9E+09,9E+09,9E+09]];
    VAR robtarget PushFilter17 := [[664.3331,-108.3433,384.4006],[0.006609402,0.4401523,0.8978986,0.0006644762],[0,0,1,0],[130.8402,9E+09,9E+09,9E+09,9E+09,9E+09]];
    VAR robtarget PushFilter18 := [[651.4076,-117.9172,384.3516],[0.006577531,0.4400893,0.8979297,0.0006210515],[1,0,1,0],[130.8029,9E+09,9E+09,9E+09,9E+09,9E+09]];
    VAR robtarget PushFilter19 := [[733.2577,-46.34735,458.0763],[0.5866504,-0.3494981,0.7297264,-0.03452196],[1,1,2,5],[170.9967,9E+09,9E+09,9E+09,9E+09,9E+09]];
    VAR robtarget PushFilter20 := [[720.921,-63.57402,380.5577],[0.02661204,-0.762087,-0.2717952,-0.5870627],[1,0,1,5],[170.9985,9E+09,9E+09,9E+09,9E+09,9E+09]];

    !points to PutUsedFilterInPlate
    VAR robtarget PutUsedFilterInPlate1 := [[473.6227,-252.2065,279.1347],[0.6325881,-0.7069083,0.292002,-0.1218517],[1,0,2,4],[-165.909,9E+09,9E+09,9E+09,9E+09,9E+09]];
    VAR robtarget PutUsedFilterInPlate2:= [[574.4794,-235.4697,49.00514],[0.4863034,-0.4829491,0.5373127,-0.4914918],[1,1,1,4],[-157.2493,9E+09,9E+09,9E+09,9E+09,9E+09]];
    VAR robtarget PutUsedFilterInPlate3 := [[514.0889,-247.6884,143.5489],[0.4872082,-0.5422345,0.4708532,-0.4968975],[1,1,1,4],[-159.2458,9E+09,9E+09,9E+09,9E+09,9E+09]];
    VAR robtarget PutUsedFilterInPlate4 := [[530.6711,-252.6093,318.137],[0.599079,-0.5827813,0.4087358,-0.3666134],[1,1,1,4],[-160.9291,9E+09,9E+09,9E+09,9E+09,9E+09]];
    VAR robtarget PutUsedFilterInPlate5 := [[391.5533,-233.6493,580.6913],[0.7759497,-0.6290888,-0.033647,-0.03189521],[1,0,2,4],[178.5084,9E+09,9E+09,9E+09,9E+09,9E+09]];
    VAR robtarget PutUsedFilterInPlate6 := [[566.8242,-237.7017,335.2878],[0.2433534,0.3150106,0.7158626,0.5736622],[1,0,0,4],[172.7277,9E+09,9E+09,9E+09,9E+09,9E+09]];
    VAR robtarget PlateInPlace := [[627.95,-154.2937,333.2767],[0.1975931,0.2695499,0.6932085,0.6385622],[1,0,0,4],[166.0525,9E+09,9E+09,9E+09,9E+09,9E+09]];

    !Points for BorderingFilterToPutInPlate
    VAR robtarget BorderingFilterToPutInPlate1 := [[675.6477,-214.1475,507.9201],[0.004738619,-0.7108954,-0.0161659,-0.7030959],[1,-2,-1,4],[175.1633,9E+09,9E+09,9E+09,9E+09,9E+09]];
    VAR robtarget BorderingFilterToPutInPlate2 := [[113.5013,-37.46609,79.09233],[0.02876629,0.7071135,-0.03476489,0.7056588],[1,-2,0,4],[127.6906,9E+09,9E+09,9E+09,9E+09,9E+09]];
    VAR robtarget BorderingFilterToPutInPlate3 := [[93.81635,6.562484,57.52491],[0.09276452,0.6824939,0.09494647,0.7187364],[1,-2,-1,4],[127.7968,9E+09,9E+09,9E+09,9E+09,9E+09]];
    VAR robtarget BorderingFilterToPutInPlate4 := [[88.22985,31.19816,53.94881],[0.07252922,0.6804215,0.1459732,0.7144634],[1,-2,0,4],[128.4669,9E+09,9E+09,9E+09,9E+09,9E+09]];
    VAR robtarget BorderingFilterToPutInPlate5 := [[77.45119,62.40168,52.68208],[0.05411451,0.6635692,0.1976721,0.7194952],[1,-2,0,4],[129.3063,9E+09,9E+09,9E+09,9E+09,9E+09]];
    VAR robtarget BorderingFilterToPutInPlate6 := [[567.22,-173.2041,316.7787],[0.2664002,0.3040051,0.6687229,0.6240364],[1,0,0,4],[-160.9951,9E+09,9E+09,9E+09,9E+09,9E+09]];

    !Points to Move plate from stack to red piece near big jar
    VAR robtarget MovePlateFromStackToRedLocation1 := [[567.22,-173.2041,316.7787],[0.2664002,0.3040051,0.6687229,0.6240364],[1,0,0,4],[-160.9951,9E+09,9E+09,9E+09,9E+09,9E+09]];
    VAR robtarget MovePlateFromStackToRedLocation2 := [[567.22,-173.2041,316.7787],[0.2664002,0.3040051,0.6687229,0.6240364],[1,0,0,4],[-160.9951,9E+09,9E+09,9E+09,9E+09,9E+09]];
    VAR robtarget MovePlateFromStackToRedLocation3 := [[567.22,-173.2041,316.7787],[0.2664002,0.3040051,0.6687229,0.6240364],[1,0,0,4],[-160.9951,9E+09,9E+09,9E+09,9E+09,9E+09]];
    VAR robtarget MovePlateFromStackToRedLocation4 := [[567.22,-173.2041,316.7787],[0.2664002,0.3040051,0.6687229,0.6240364],[1,0,0,4],[-160.9951,9E+09,9E+09,9E+09,9E+09,9E+09]];
    VAR robtarget MovePlateFromStackToRedLocation5 := [[567.22,-173.2041,316.7787],[0.2664002,0.3040051,0.6687229,0.6240364],[1,0,0,4],[-160.9951,9E+09,9E+09,9E+09,9E+09,9E+09]];
    VAR robtarget MovePlateFromStackToRedLocation6 := [[567.22,-173.2041,316.7787],[0.2664002,0.3040051,0.6687229,0.6240364],[1,0,0,4],[-160.9951,9E+09,9E+09,9E+09,9E+09,9E+09]];
    VAR robtarget MovePlateFromStackToRedLocation7 := [[567.22,-173.2041,316.7787],[0.2664002,0.3040051,0.6687229,0.6240364],[1,0,0,4],[-160.9951,9E+09,9E+09,9E+09,9E+09,9E+09]];
    VAR robtarget MovePlateFromStackToRedLocation8 := [[567.22,-173.2041,316.7787],[0.2664002,0.3040051,0.6687229,0.6240364],[1,0,0,4],[-160.9951,9E+09,9E+09,9E+09,9E+09,9E+09]];

    ! Some points to pick the plate
    VAR robtarget PickPlate1 := [[227.1261,-527.5699,341.0041],[0.04053182,-0.8623218,-0.4814033,0.1516877],[0,-1,1,4],[176.1331,9E+09,9E+09,9E+09,9E+09,9E+09]];
    VAR robtarget PickPlate2 := [[-3.567228,-408.2107,134.7796],[0.3952619,-0.6121742,-0.4965889,0.471604],[0,-1,1,4],[-130.3624,9E+09,9E+09,9E+09,9E+09,9E+09]];
    VAR robtarget PickPlate3 := [[-142.6978,-318.9195,42.63297],[0.4808339,-0.4860117,-0.518315,0.5137518],[1,-1,1,4],[-143.24,9E+09,9E+09,9E+09,9E+09,9E+09]];
    VAR robtarget PickPlate4 := [[-142.4758,-318.8727,61.93118],[0.4808406,-0.4865499,-0.5182256,0.5133262],[1,-1,1,4],[-143.2737,9E+09,9E+09,9E+09,9E+09,9E+09]];
    VAR robtarget PickPlate5 := [[-77.97506,-326.9365,96.9474],[0.5010442,-0.5218936,-0.4985341,0.4775413],[0,-1,1,4],[-136.8395,9E+09,9E+09,9E+09,9E+09,9E+09]];
    VAR robtarget PickPlate6 := [[-90.30951,-320.5932,44.24039],[0.4979136,-0.5123259,-0.5073266,0.4818961],[1,-1,1,4],[-143.0363,9E+09,9E+09,9E+09,9E+09,9E+09]];
    VAR robtarget PickPlate7 := [[-61.84347,-321.6961,44.76805],[0.4966117,-0.5100227,-0.50834,0.4846072],[1,-1,1,4],[-142.9827,9E+09,9E+09,9E+09,9E+09,9E+09]];
    VAR robtarget PickPlate8 := [[-52.97003,-322.5573,106.2267],[0.4950693,-0.5096297,-0.5090222,0.485881],[0,-1,1,4],[-142.9297,9E+09,9E+09,9E+09,9E+09,9E+09]];
    VAR robtarget PickPlate9 := [[-44.28172,-319.6465,128.838],[0.6372106,-0.3134488,-0.6291855,-0.3159717],[0,-1,0,4],[-133.2934,9E+09,9E+09,9E+09,9E+09,9E+09]];
    VAR robtarget PickPlate10_1 := [[-143.5759,-241.5467,111.6477],[0.6093763,-0.4017231,-0.5714734,-0.3750964],[0,-1,0,4],[-141.1836,9E+09,9E+09,9E+09,9E+09,9E+09]];
    VAR robtarget PickPlate10_2 := [[-167.7915,-241.5351,118.1164],[0.6093708,-0.4017192,-0.571467,-0.3751193],[0,-1,0,4],[-141.1944,9E+09,9E+09,9E+09,9E+09,9E+09]];
    VAR robtarget PickPlate10_3 := [[-167.7915,-241.5351,123.1164],[0.6093708,-0.4017192,-0.571467,-0.3751193],[0,-1,0,4],[-141.1944,9E+09,9E+09,9E+09,9E+09,9E+09]];
    VAR robtarget PickPlate10_4 := [[-37.56079,-321.5652,103.587],[0.547386,-0.3171856,-0.6532114,-0.416025],[1,-1,0,4],[-144.1172,9E+09,9E+09,9E+09,9E+09,9E+09]];
    VAR robtarget PickPlate11_Down := [[-143.5759,-241.5467,134.8745],[0.6093763,-0.4017231,-0.5714734,-0.3750964],[0,-1,0,4],[-141.1836,9E+09,9E+09,9E+09,9E+09,9E+09]];
    VAR robtarget PickPlate11_Up := [[-143.5759,-241.5467,134.8745],[0.6093763,-0.4017231,-0.5714734,-0.3750964],[0,-1,0,4],[-141.1836,9E+09,9E+09,9E+09,9E+09,9E+09]];
    VAR robtarget PickPlate12 := [[-241.0147,-241.6081,137.761],[0.616179,-0.391013,-0.5779745,-0.3652091],[0,-1,0,4],[-141.1788,9E+09,9E+09,9E+09,9E+09,9E+09]];
    VAR robtarget PickPlate13 := [[-241.1691,-241.7823,111.6477],[0.6093817,-0.4017254,-0.5714735,-0.3750848],[1,-1,0,4],[-141.1598,9E+09,9E+09,9E+09,9E+09,9E+09]];
    VAR robtarget PickPlate14_ThrowPlateCover := [[-74.80486,-257.3926,223.272],[0.5064288,-0.4275604,-0.5680993,-0.4878372],[0,0,0,4],[-151.8755,9E+09,9E+09,9E+09,9E+09,9E+09]];

    ! Some points to put plate in Capinet

    VAR robtarget PutPlateInCapinet1PreMoving := [[622.3975,-163.4876,346.3798],[0.2100825,0.2565895,0.7139377,0.616701],[1,0,0,4],[161.9459,9E+09,9E+09,9E+09,9E+09,9E+09]];
    VAR robtarget PutPlateInCapinet1 := [[336.9954,-126.1508,641.6207],[0.2318186,0.05682539,-0.6800953,-0.6931821],[1,0,1,4],[-162.4004,9E+09,9E+09,9E+09,9E+09,9E+09]];
    VAR robtarget PutPlateInCapinet2 := [[107.7427,-67.06541,778.0781],[0.3994297,0.347616,-0.6359779,-0.5613832],[1,0,1,4],[-121.987,9E+09,9E+09,9E+09,9E+09,9E+09]];
    VAR robtarget PutPlateInCapinet3 := [[-39.04373,-73.9049,744.7962],[0.4666459,0.476293,-0.5254644,-0.5284635],[1,0,1,4],[-116.1677,9E+09,9E+09,9E+09,9E+09,9E+09]];
    VAR robtarget PutPlateInCapinet4 := [[23.16677,-73.90886,713.7164],[0.4666705,0.4762923,-0.5254518,-0.5284551],[1,0,1,4],[-116.1661,9E+09,9E+09,9E+09,9E+09,9E+09]];
    VAR robtarget PutPlateInCapinet5 := [[-39.03989,-73.90785,713.7233],[0.466655,0.476292,-0.5254535,-0.5284672],[1,0,1,4],[-116.1664,9E+09,9E+09,9E+09,9E+09,9E+09]];
    VAR robtarget PutPlateInCapinet6 := [[-37.01698,-73.91552,761.9521],[0.466686,0.4762945,-0.5254425,-0.5284486],[1,0,1,4],[-116.1639,9E+09,9E+09,9E+09,9E+09,9E+09]];
    VAR robtarget PutPlateInCapinet7 := [[-212.6318,-334.0861,481.3083],[0.6006479,-0.400857,-0.606375,-0.3329342],[0,-1,-1,4],[-113.8211,9E+09,9E+09,9E+09,9E+09,9E+09]];
    VAR robtarget PutPlateInCapinet8 := [[-212.6318,-334.0861,481.3083],[0.6006479,-0.400857,-0.606375,-0.3329342],[0,-1,-1,4],[-113.8211,9E+09,9E+09,9E+09,9E+09,9E+09]];
    VAR robtarget PutPlateInCapinet9 := [[-212.6318,-334.0861,481.3083],[0.6006479,-0.400857,-0.606375,-0.3329342],[0,-1,-1,4],[-113.8211,9E+09,9E+09,9E+09,9E+09,9E+09]];

    !points to take out the plate from the closet

    VAR robtarget AbovePlateInCloset := [[-37.01698,-73.91552,791.9521],[0.466686,0.4762945,-0.5254425,-0.5284486],[1,0,1,4],[-116.1639,9E+09,9E+09,9E+09,9E+09,9E+09]];
    VAR robtarget AroundPlateInCloset := [[-36.92104,-73.94338,713.5489],[0.466785,0.4762551,-0.5253302,-0.5285084],[1,0,1,4],[-116.1534,9E+09,9E+09,9E+09,9E+09,9E+09]];
    VAR robtarget TakePlateOut1 := [[153.3338,-128.2487,793.0741],[0.4162462,0.5471437,-0.473133,-0.5509248],[1,0,1,4],[-119.9038,9E+09,9E+09,9E+09,9E+09,9E+09]];
    VAR robtarget TakePlateOut2 := [[653.3688,-154.808,526.8815],[0.1977761,0.3044988,0.6442697,0.6731133],[1,-1,1,4],[-155.923,9E+09,9E+09,9E+09,9E+09,9E+09]];
    VAR robtarget PlateAboveBigJar := [[666.7081,-111.3742,401.4151],[0.2972408,0.3367108,0.6372746,0.6262226],[1,-1,1,4],[-165.2874,9E+09,9E+09,9E+09,9E+09,9E+09]];
    VAR robtarget PlateOnBigJar := [[666.7331,-111.2638,365.1944],[0.2982312,0.3357119,0.6368653,0.6267043],[1,-1,1,4],[-165.2628,9E+09,9E+09,9E+09,9E+09,9E+09]];
    VAR robtarget PlateOnBigJar1 := [[666.7374,-111.2572,359.6436],[0.2982137,0.3356809,0.6368814,0.6267129],[1,0,0,4],[-165.2619,9E+09,9E+09,9E+09,9E+09,9E+09]];


    !Points tp pick the filter for analysis
    VAR robtarget PickFilterForAnalysis1 := [[675.5394,-108.0748,503.7346],[0.6090953,-0.2344455,0.7329304,0.1919672],[1,-1,0,4],[-175.308,9E+09,9E+09,9E+09,9E+09,9E+09]];
    VAR robtarget AboveFilterForAnalysis := [[718.9147,-65.57491,471.2317],[0.6941316,-0.2419525,0.6493869,0.1947739],[1,-1,0,5],[170.0938,9E+09,9E+09,9E+09,9E+09,9E+09]];
    VAR robtarget PickFilterForAnalysis := [[732.3462,-74.86136,412.2591],[0.6741185,-0.220105,0.6811666,0.1820167],[1,-1,0,5],[166.8679,9E+09,9E+09,9E+09,9E+09,9E+09]];


   !poibnts to remove the plate after the analysis
    VAR robtarget MovePlateAfterAnalysis1 := [[732.3462,-74.86136,412.2591],[0.6741185,-0.220105,0.6811666,0.1820167],[1,-1,0,5],[166.8679,9E+09,9E+09,9E+09,9E+09,9E+09]];
    VAR robtarget MovePlateAfterAnalysis2 := [[732.3462,-74.86136,412.2591],[0.6741185,-0.220105,0.6811666,0.1820167],[1,-1,0,5],[166.8679,9E+09,9E+09,9E+09,9E+09,9E+09]];
    VAR robtarget MovePlateAfterAnalysis3 := [[663.5577,-116.3641,387.2455],[0.02010107,0.574471,0.818178,0.01280024],[0,-1,1,0],[140.1178,9E+09,9E+09,9E+09,9E+09,9E+09]];
    VAR robtarget MovePlateAfterAnalysis4 := [[663.5488,-116.4332,398.0156],[0.02007263,0.5745333,0.8181344,0.0128338],[0,-1,1,0],[140.1235,9E+09,9E+09,9E+09,9E+09,9E+09]];
    VAR robtarget MovePlateAfterAnalysis5 := [[462.5022,-435.4173,392.7523],[0.02093044,0.6087145,0.792644,0.02727618],[0,-1,1,4],[140.0694,9E+09,9E+09,9E+09,9E+09,9E+09]];
    VAR robtarget MovePlateAfterAnalysis6 := [[484.446,-345.5098,107.2954],[0.05076824,-0.699346,-0.7125604,-0.02440064],[1,-1,1,4],[156.0081,9E+09,9E+09,9E+09,9E+09,9E+09]];
    VAR robtarget MovePlateAfterAnalysis7 := [[462.8721,-336.8476,46.51273],[0.03607976,-0.6682198,-0.7430834,-0.002757301],[1,-1,1,4],[154.5291,9E+09,9E+09,9E+09,9E+09,9E+09]];



    !Points to CloseCapinet
    VAR robtarget CloseCapinet1 := [[207.5222,-242.1754,591.3132],[0.06543734,-0.0622346,-0.6650254,-0.7413408],[1,0,1,4],[-170.9305,9E+09,9E+09,9E+09,9E+09,9E+09]];
    VAR robtarget CloseCapinet2 := [[-22.68939,-315.5607,560.8279],[0.2878203,-0.207479,-0.611744,-0.7070227],[1,0,2,4],[102.4968,9E+09,9E+09,9E+09,9E+09,9E+09]];
    VAR robtarget CloseCapinet3 := [[-120.784,-345.9569,597.4397],[0.3498625,0.001832771,-0.5227011,-0.7774165],[1,1,2,4],[98.65139,9E+09,9E+09,9E+09,9E+09,9E+09]];
    VAR robtarget CloseCapinet4 := [[-82.97842,-382.2726,644.6324],[0.03086359,-0.1110591,0.3303497,0.9367937],[1,0,1,4],[98.49933,9E+09,9E+09,9E+09,9E+09,9E+09]];
    VAR robtarget CloseCapinet5 := [[-33.28422,-393.3404,662.8998],[0.05534496,-0.08431086,-0.2613863,-0.9599509],[1,0,1,4],[100.3842,9E+09,9E+09,9E+09,9E+09,9E+09]];
    VAR robtarget CloseCapinet6 := [[126.8073,-299.3019,691.0593],[0.1787152,-0.2536302,-0.5090077,-0.8028972],[1,0,1,4],[166.1153,9E+09,9E+09,9E+09,9E+09,9E+09]];
    VAR robtarget CloseCapinet7 := [[195.0965,-120.0588,719.5216],[0.4439963,-0.1593523,-0.7213333,-0.507102],[1,0,1,4],[-150.4515,9E+09,9E+09,9E+09,9E+09,9E+09]];
    VAR robtarget CloseCapinet8 := [[96.39011,-1.393748,742.2653],[0.5350459,-0.062455,-0.7222924,-0.4337268],[1,0,1,4],[-138.2767,9E+09,9E+09,9E+09,9E+09,9E+09]];
    VAR robtarget CloseCapinet9 := [[63.36932,10.57348,768.642],[0.6800932,-0.05562977,-0.7297705,-0.04258671],[1,0,2,4],[-133.4059,9E+09,9E+09,9E+09,9E+09,9E+09]];
    VAR robtarget CloseCapinet10 := [[52.19879,11.1265,767.5461],[0.6809717,-0.0249305,-0.7318537,-0.006795681],[1,0,1,4],[-132.5736,9E+09,9E+09,9E+09,9E+09,9E+09]];

    VAR robtarget MoveDispenser1 := [[382.0439,-119.625,292.9677],[0.7184659,-0.6954051,0.002741368,0.01452396],[0,1,1,4],[107.1018,9E+09,9E+09,9E+09,9E+09,9E+09]];
    VAR robtarget MoveDispenser2 := [[367.2742,-97.70506,472.0224],[0.7114094,-0.7025003,0.004124381,-0.0193076],[0,0,2,4],[137.8868,9E+09,9E+09,9E+09,9E+09,9E+09]];
    VAR robtarget MoveDispenser3 := [[296.933,-82.52208,478.6049],[0.7070982,-0.7064348,0.02777747,-0.01379868],[0,0,2,4],[145.1462,9E+09,9E+09,9E+09,9E+09,9E+09]];
    VAR robtarget MoveDispenser31 := [[296.933,-98.82317,447.6208],[0.705121,-0.7090259,0.003036739,-0.008797801],[0,0,2,4],[148.4961,9E+09,9E+09,9E+09,9E+09,9E+09]];
    VAR robtarget MoveDispenser4 := [[296.933,-113.715,419.1608],[0.7027627,-0.7111467,-0.01941378,-0.004263762],[0,0,2,4],[151.5516,9E+09,9E+09,9E+09,9E+09,9E+09]];
    VAR robtarget MoveDispenser5 := [[296.933,-135.4433,412.0101],[0.7132996,-0.7001655,0.0264315,-0.01653659],[0,0,1,4],[124.0881,9E+09,9E+09,9E+09,9E+09,9E+09]];
    VAR robtarget MoveDispenser6_1 := [[296.9357,-144.6807,396.5883],[0.7462527,-0.665211,0.02072768,-0.0131015],[0,0,2,4],[167.538,9E+09,9E+09,9E+09,9E+09,9E+09]];
    VAR robtarget MoveDispenser6_2 := [[296.9381,-144.6735,396.579],[0.727263,-0.685921,0.02034875,-0.01366454],[0,0,2,4],[167.5494,9E+09,9E+09,9E+09,9E+09,9E+09]];
    VAR robtarget MoveDispenser7 := [[295.9322,-206.0766,442.1875],[0.7091605,-0.7050132,0.005624216,0.004032394],[0,0,2,4],[138.4178,9E+09,9E+09,9E+09,9E+09,9E+09]];
    VAR robtarget MoveDispenser8 := [[316.067,-25.3562,539.6172],[0.5164476,-0.4981974,0.4920629,0.492905],[0,1,3,4],[114.3105,9E+09,9E+09,9E+09,9E+09,9E+09]];
    VAR robtarget MoveDispenser9 := [[324.9807,-24.98611,513.7685],[0.4891407,-0.4735606,0.5265107,0.5091838],[0,1,3,4],[118.2191,9E+09,9E+09,9E+09,9E+09,9E+09]];
    VAR robtarget MoveDispenser10 := [[325.1716,-25.00177,494.9056],[0.4893806,-0.4731246,0.5266935,0.5091697],[0,1,2,4],[113.0836,9E+09,9E+09,9E+09,9E+09,9E+09]];
    VAR robtarget MoveDispenser10Clear := [[325.1701,-25.00095,491.0015],[0.4893791,-0.4731236,0.526693,0.5091724],[0,1,2,4],[113.0846,9E+09,9E+09,9E+09,9E+09,9E+09]];
    VAR robtarget MoveDispenser11 := [[292.933,-189.7269,398.1999],[0.7107903,-0.7032589,0.01307814,0.005744404],[0,0,1,4],[140.9083,9E+09,9E+09,9E+09,9E+09,9E+09]];
    VAR robtarget MoveDispenser12 := [[296.933,-133.6059,398.1976],[0.7107857,-0.7032634,0.01308545,0.005749269],[0,0,1,4],[140.8967,9E+09,9E+09,9E+09,9E+09,9E+09]];

    ! Points to ensure Tight Equipment of the nozzle
    VAR robtarget TightEquipping_1 := [[535.3924,-105.5459,384.5103],[0.7103947,-0.6961535,0.07582311,-0.07043169],[0,1,1,4],[105.5924,9E+09,9E+09,9E+09,9E+09,9E+09]];
    VAR robtarget TightEquipping_2 := [[535.3889,-105.5355,300.3238],[0.710388,-0.6961632,0.07581223,-0.07041441],[1,1,1,4],[105.5948,9E+09,9E+09,9E+09,9E+09,9E+09]];
    VAR robtarget TightEquipping_2_2 := [[535.3889,-105.5355,288.8238],[0.710388,-0.6961632,0.07581223,-0.07041441],[1,1,1,4],[105.5948,9E+09,9E+09,9E+09,9E+09,9E+09]];
    VAR robtarget TightEquipping_3_1 := [[354.7574,-419.8932,481.9371],[0.5413219,-0.5402309,0.4912076,-0.4169367],[0,1,1,4],[48.37782,9E+09,9E+09,9E+09,9E+09,9E+09]];
    VAR robtarget TightEquipping_3_2 := [[481.5215,-314.9106,527.3628],[0.6543044,-0.6797594,0.2464043,-0.2215801],[0,1,2,4],[96.73737,9E+09,9E+09,9E+09,9E+09,9E+09]];

    !points TO move filter FOR analysis
    VAR robtarget MoveFilterForAnalysis1 := [[576.2863,-266.4957,300.7272],[0.5131347,-0.8375504,0.03206132,-0.1848626],[1,1,1,4],[83.75623,9E+09,9E+09,9E+09,9E+09,9E+09]];
    VAR robtarget MoveFilterForAnalysis2 := [[551.3336,-141.4326,496.0421],[0.5076712,-0.4920709,0.6933403,0.139339],[0,-2,1,5],[137.2368,9E+09,9E+09,9E+09,9E+09,9E+09]];
    VAR robtarget MoveFilterForAnalysis3 := [[670.7968,-216.9672,476.6045],[0.6567829,-0.1226356,0.7438014,-0.01887434],[0,-2,1,4],[164.5108,9E+09,9E+09,9E+09,9E+09,9E+09]];
    VAR robtarget MoveFilterForAnalysis4 := [[571.4567,-387.3068,421.7431],[0.5294378,-0.0225638,0.8479175,-0.01491239],[0,-2,1,4],[138.8005,9E+09,9E+09,9E+09,9E+09,9E+09]];
    VAR robtarget MoveFilterForAnalysis5 := [[423.464,-575.4677,360.5327],[0.4773839,0.2307418,0.8379274,-0.1293854],[0,-2,1,4],[146.3012,9E+09,9E+09,9E+09,9E+09,9E+09]];
    VAR robtarget MoveFilterForAnalysis6 := [[193.5765,-566.7524,271.4265],[0.2991756,0.1483591,0.7243653,-0.6031405],[0,-2,1,4],[-150.8147,9E+09,9E+09,9E+09,9E+09,9E+09]];
    VAR robtarget MoveFilterForAnalysis7 := [[-29.78449,-564.9139,203.7348],[0.07294004,0.03285255,0.687743,-0.7215331],[0,-2,1,4],[-136.5771,9E+09,9E+09,9E+09,9E+09,9E+09]];
    VAR robtarget MoveFilterForAnalysis8 := [[-60.96145,-570.5043,102.7206],[0.0003970733,0.0003768174,-0.7069172,0.7072961],[0,-2,1,4],[-136.6732,9E+09,9E+09,9E+09,9E+09,9E+09]];
    VAR robtarget MoveFilterForAnalysis9 := [[-60.95448,-570.4955,76.06806],[0.000390227,0.000370277,-0.7069259,0.7072874],[1,-2,1,4],[-136.6796,9E+09,9E+09,9E+09,9E+09,9E+09]];




    !points to move tube from red station to analysis jars


    VAR robtarget MoveJarFromRedStation2analysis1 := [[505.6292,-223.0625,343.9532],[0.6722786,-0.7395206,0.02152137,-0.0262216],[0,1,1,4],[108.8755,9E+09,9E+09,9E+09,9E+09,9E+09]];
    VAR robtarget MoveJarFromRedStation2analysis2 := [[546.0399,-115.6157,170.9639],[0.676777,-0.7360623,0.01360704,9.801232E-05],[1,0,1,4],[141.0371,9E+09,9E+09,9E+09,9E+09,9E+09]];
    VAR robtarget MoveJarFromRedStation2analysis3 := [[539.332,-75.38523,181.0287],[0.6922007,-0.7194945,0.04406742,-0.0352692],[1,0,1,4],[152.1927,9E+09,9E+09,9E+09,9E+09,9E+09]];
    VAR robtarget MoveJarFromRedStation2analysis4 := [[539.3273,-75.38727,94.37062],[0.6921986,-0.7194971,0.04406229,-0.03526428],[1,0,1,4],[152.1915,9E+09,9E+09,9E+09,9E+09,9E+09]];
    VAR robtarget MoveJarFromRedStation2analysis5 := [[522.342,-334.9005,241.1796],[0.6052258,-0.5608471,0.4194907,-0.3783911],[0,1,1,4],[141.4391,9E+09,9E+09,9E+09,9E+09,9E+09]];
    VAR robtarget MoveJarFromRedStation2analysis6 := [[113.6483,-487.3515,250.8779],[0.4180533,-0.4069934,-0.5550178,0.5929107],[0,3,1,4],[147.779,9E+09,9E+09,9E+09,9E+09,9E+09]];
    VAR robtarget MoveJarFromRedStation2analysis7 := [[-19.71465,-445.9225,226.1846],[0.5164229,-0.4576384,-0.5229003,0.5004495],[0,3,1,4],[171.6785,9E+09,9E+09,9E+09,9E+09,9E+09]];
    VAR robtarget MoveJarFromRedStation2analysis8 := [[-179.1799,-420.765,158.0618],[0.4901585,-0.5050656,-0.5158308,0.4884383],[0,3,1,4],[-139.8235,9E+09,9E+09,9E+09,9E+09,9E+09]];
    VAR robtarget MoveJarFromRedStation2analysis9 := [[-179.1564,-420.7976,158.0813],[0.6326635,-0.2860823,-0.6628262,0.280277],[0,3,1,4],[-139.8259,9E+09,9E+09,9E+09,9E+09,9E+09]];
    VAR robtarget MoveJarFromRedStation2analysis10 := [[-177.9918,-455.98,133.8936],[0.6788174,0.1239778,-0.7144292,-0.1158763],[0,3,0,4],[-143.9907,9E+09,9E+09,9E+09,9E+09,9E+09]];
    !Increased z+10
    VAR robtarget MoveJarFromRedStation2Moving1 := [[-84.72699,-431.0913,124.4718],[0.4975998,-0.4967284,-0.5026339,0.5030055],[0,3,1,4],[-147.9485,9E+09,9E+09,9E+09,9E+09,9E+09]];
    VAR robtarget MoveJarFromRedStation2Moving2 := [[-84.72606,-455.5026,115.5713],[0.505415,-0.4887927,-0.5103554,0.4951511],[0,3,1,4],[-147.9649,9E+09,9E+09,9E+09,9E+09,9E+09]];
    VAR robtarget MoveJarFromRedStation2Moving3 := [[-84.72516,-455.5017,115.5705],[0.7070269,0.03500611,-0.7058017,-0.02704729],[0,3,0,4],[-147.9615,9E+09,9E+09,9E+09,9E+09,9E+09]];



    !points to drag station on rails
    VAR robtarget DragRailStation1 := [[-181.9899,-440.7072,200.4893],[0.5101894,-0.4819916,-0.4901209,0.5168873],[0,3,1,4],[-150.8767,9E+09,9E+09,9E+09,9E+09,9E+09]];
    VAR robtarget DragRailStation2 := [[-234.1095,-444.6271,190.0733],[0.5047785,-0.4705801,-0.5122988,0.511178],[0,3,1,4],[-147.3724,9E+09,9E+09,9E+09,9E+09,9E+09]];
    VAR robtarget DragRailStation3 := [[-170.8042,-445.1068,190.7449],[0.5073108,-0.4954348,-0.5010529,0.496111],[0,3,1,4],[-157.8092,9E+09,9E+09,9E+09,9E+09,9E+09]];
    VAR robtarget DragRailStation4 := [[-77.57322,-443.454,185.8936],[0.5149699,-0.4874528,-0.4917896,0.5053106],[0,3,1,4],[-147.4562,9E+09,9E+09,9E+09,9E+09,9E+09]];
    VAR robtarget DragRailStation5 := [[21.82821,-420.2001,202.8728],[0.5002174,-0.4939232,-0.5112581,0.4944063],[0,3,1,4],[-153.442,9E+09,9E+09,9E+09,9E+09,9E+09]];
    VAR robtarget DragRailStation6 := [[-122.9713,-440.1708,178.95],[0.4771074,-0.5249177,-0.5113651,0.485114],[0,3,1,4],[-151.1015,9E+09,9E+09,9E+09,9E+09,9E+09]];
    VAR robtarget DragRailStation7 := [[-73.14442,-441.7872,183.3839],[0.5046592,-0.5173727,-0.4904874,0.4868949],[0,3,1,4],[-149.047,9E+09,9E+09,9E+09,9E+09,9E+09]];


    !Ponints to push station on rails
    VAR robtarget PushRailStation1 := [[283.519,-537.2913,301.1427],[0.1730787,0.813297,-0.520491,-0.1941154],[0,0,2,4],[103.529,9E+09,9E+09,9E+09,9E+09,9E+09]];
    VAR robtarget PushRailStation2 := [[61.73232,-422.8468,229.6872],[0.41526,-0.5235382,-0.4602712,0.5844804],[0,-1,1,4],[168.0418,9E+09,9E+09,9E+09,9E+09,9E+09]];
    VAR robtarget PushRailStation3 := [[-30.17656,-453.6681,190.053],[0.4731088,-0.5148413,-0.5033177,0.5077183],[0,-1,1,4],[172.7681,9E+09,9E+09,9E+09,9E+09,9E+09]];
    VAR robtarget PushRailStation4 := [[-126.3609,-453.6584,190.0475],[0.4731194,-0.5148572,-0.5033104,0.5076994],[1,-1,1,4],[172.7693,9E+09,9E+09,9E+09,9E+09,9E+09]];
    VAR robtarget PushRailStation5 := [[-176.1112,-453.6546,190.0476],[0.4731254,-0.5148618,-0.5033034,0.5076962],[1,-1,1,4],[172.7673,9E+09,9E+09,9E+09,9E+09,9E+09]];
    VAR robtarget PushRailStation6 := [[-192.4105,-453.6254,190.0467],[0.4731468,-0.5148733,-0.5032885,0.5076793],[1,-1,1,4],[172.7641,9E+09,9E+09,9E+09,9E+09,9E+09]];


    !Point to pick Weird Jar
    VAR robtarget PickWeirdJar1 := [[438.673,-264.6234,436.7415],[0.1032414,-0.4197006,-0.86777,-0.2452915],[0,-1,1,4],[168.2663,9E+09,9E+09,9E+09,9E+09,9E+09]];
    VAR robtarget PickWeirdJar2 := [[422.3206,-414.3522,286.8045],[0.06316473,-0.8432161,-0.5320243,0.0441245],[0,0,1,4],[122.607,9E+09,9E+09,9E+09,9E+09,9E+09]];
    VAR robtarget PickWeirdJar3 := [[464.9016,-440.0679,189.7729],[0.004917408,-0.9984844,0.03392469,0.04305722],[0,0,2,4],[106.7649,9E+09,9E+09,9E+09,9E+09,9E+09]];
    VAR robtarget AboveWeirdJar := [[463.6422,-449.7212,181.5877],[0.1965588,0.9803609,-0.01538027,0.004534668],[0,-1,2,4],[126.7406,9E+09,9E+09,9E+09,9E+09,9E+09]];
    VAR robtarget AroundWeirdJar := [[463.6242,-465.1023,144.824],[0.196559,0.9803612,-0.01536489,0.004512812],[1,-1,2,4],[126.7383,9E+09,9E+09,9E+09,9E+09,9E+09]];

    !Points to place stationary weird jar
    VAR robtarget PlaceStatinaryWeirdJar1 := [[252.4259,-480.2196,321.9088],[0.02096372,-0.9850105,-0.1708974,0.01043308],[0,0,1,4],[86.11672,9E+09,9E+09,9E+09,9E+09,9E+09]];
    VAR robtarget PlaceStatinaryWeirdJar2 := [[12.92549,-488.528,288.3879],[0.01863053,-0.9980026,0.06012812,-0.005318572],[0,0,1,4],[-102.0417,9E+09,9E+09,9E+09,9E+09,9E+09]];
    VAR robtarget PlaceStatinaryWeirdJar3 := [[-96.23866,-498.9594,179.6048],[0.00874308,0.9988055,-0.04805301,-0.001441678],[0,0,1,4],[-119.849,9E+09,9E+09,9E+09,9E+09,9E+09]];
    VAR robtarget AboveStationary := [[-167.8721,-493.7102,154.5018],[0.001056325,0.9995645,-0.02947625,0.0009529712],[0,0,1,4],[-111.6589,9E+09,9E+09,9E+09,9E+09,9E+09]];
    VAR robtarget InStationary := [[-167.8714,-493.7118,113.946],[0.001058074,0.9995645,-0.02947489,0.0009530607],[0,0,1,4],[-111.6724,9E+09,9E+09,9E+09,9E+09,9E+09]];

!Points to place moving weird jar
    VAR robtarget PlaceMovingWeirdJar1 := [[252.4259,-480.2196,321.9088],[0.02096372,-0.9850105,-0.1708974,0.01043308],[0,0,1,4],[86.11672,9E+09,9E+09,9E+09,9E+09,9E+09]];
    VAR robtarget PlaceMovingWeirdJar2 := [[167.2292,-476.5943,231.9351],[0.03677763,-0.649482,-0.7593842,0.01250212],[0,0,0,4],[159.4192,9E+09,9E+09,9E+09,9E+09,9E+09]];
    VAR robtarget PlaceMovingWeirdJar3 := [[113.8516,-495.526,188.0661],[0.0139544,-0.32726,-0.9447033,-0.01554803],[0,-1,0,4],[-147.3213,9E+09,9E+09,9E+09,9E+09,9E+09]];
    VAR robtarget AboveMoving := [[87.03879,-497.7999,162.1266],[0.0001936294,0.01576547,0.9998757,3.247788E-05],[0,0,-1,4],[-147.4099,9E+09,9E+09,9E+09,9E+09,9E+09]];
    VAR robtarget InMoving := [[87.03879,-497.7999,115.105],[0.0002035065,0.01575143,0.9998759,5.529984E-05],[0,0,-1,4],[-147.4308,9E+09,9E+09,9E+09,9E+09,9E+09]];

    !points to move pippet to stationary analysis stand
    VAR robtarget MovePippetToStationary1 := [[507.6341,-189.0893,440.8772],[0.651014,-0.6995967,0.1947547,-0.2209432],[0,1,1,4],[128.0173,9E+09,9E+09,9E+09,9E+09,9E+09]];
    VAR robtarget MovePippetToStationary2 := [[412.1312,-362.4122,453.5109],[0.5378951,-0.5284167,0.4455742,-0.4826057],[0,1,1,4],[101.7338,9E+09,9E+09,9E+09,9E+09,9E+09]];
    VAR robtarget MovePippetToStationary2_2 := [[315.248,-469.0392,463.2877],[0.3619739,-0.3388882,0.6075381,-0.6205056],[0,1,1,4],[86.00907,9E+09,9E+09,9E+09,9E+09,9E+09]];
    VAR robtarget MovePippetToStationary3 := [[90.37859,-495.4496,432.4385],[0.01336378,0.009962968,0.7073407,-0.7066762],[0,2,1,4],[-144.8657,9E+09,9E+09,9E+09,9E+09,9E+09]];
    VAR robtarget MovePippetToStationary4 := [[3.216545,-495.4931,402.0049],[0.01327836,0.01006019,0.7071336,-0.7068837],[0,2,1,4],[-137.6765,9E+09,9E+09,9E+09,9E+09,9E+09]];
    VAR robtarget MovePippetToStationary5 := [[-179.6787,-494.8793,381.61],[0.01327774,0.01004041,0.7071286,-0.7068889],[0,2,1,4],[-137.6557,9E+09,9E+09,9E+09,9E+09,9E+09]];
    VAR robtarget MovePippetToStationary6 := [[-176.874,-472.602,379.1972],[0.004065976,-0.007739501,0.7056615,-0.7084951],[0,2,1,4],[-137.2728,9E+09,9E+09,9E+09,9E+09,9E+09]];
    VAR robtarget MovePippetToStationary7 := [[-176.4472,-457.5461,337.3389],[0.000614215,0.008246354,0.6899651,-0.7237954],[0,2,1,4],[-135.1573,9E+09,9E+09,9E+09,9E+09,9E+09]];

    !Ponts to full from stationary analysis jar
    VAR robtarget FillFromStationary1 := [[-179.6764,-466.2258,432.9553],[0.01327973,0.01005142,0.7071229,-0.7068945],[0,2,2,4],[-133.7982,9E+09,9E+09,9E+09,9E+09,9E+09]];
    VAR robtarget FillFromStationary_AbovePippet := [[-268.1166,-464.8811,466.6767],[0.004425052,-0.6988553,1.853E-05,0.7152493],[0,3,2,4],[-104.8425,9E+09,9E+09,9E+09,9E+09,9E+09]];
    VAR robtarget FillFromStationary3 := [[-268.1146,-464.8816,438.9795],[0.00442743,-0.698855,1.38721E-05,0.7152497],[0,3,2,4],[-104.8602,9E+09,9E+09,9E+09,9E+09,9E+09]];
    VAR robtarget FillFromStationary4 := [[-179.6848,-466.2216,337.4254],[0.01326209,0.01003572,0.7071167,-0.7069012],[0,2,1,4],[-137.6343,9E+09,9E+09,9E+09,9E+09,9E+09]];
    VAR robtarget FillFromStationary5 := [[-179.6848,-466.2216,337.4254],[0.01326209,0.01003572,0.7071167,-0.7069012],[0,2,1,4],[-137.6343,9E+09,9E+09,9E+09,9E+09,9E+09]];
    VAR robtarget FillFromStationary6 := [[-179.6848,-466.2216,337.4254],[0.01326209,0.01003572,0.7071167,-0.7069012],[0,2,1,4],[-137.6343,9E+09,9E+09,9E+09,9E+09,9E+09]];
    !pints to move pippet to moving analysis stand
    VAR robtarget MovePippetToMoving5 := [[-92.05513,-495.495,401.9868],[0.01327694,0.01011909,0.7071326,-0.7068838],[0,2,1,4],[-137.6954,9E+09,9E+09,9E+09,9E+09,9E+09]];
    VAR robtarget MovePippetToMoving6 := [[-92.04644,-466.0188,380.2943],[0.01328323,0.01011669,0.70714,-0.7068764],[0,2,1,4],[-137.7378,9E+09,9E+09,9E+09,9E+09,9E+09]];
    VAR robtarget MovePippetToMoving7 := [[-88.24129,-463.4341,337.2401],[0.006473252,0.009628383,-0.6990232,0.7150048],[0,2,1,4],[-137.5185,9E+09,9E+09,9E+09,9E+09,9E+09]];


    VAR robtarget FillFromMoving1 := [[-88.03726,-465.0193,432.0527],[0.006473252,0.009628383,-0.6990232,0.7150048],[0,2,1,4],[-137.5185,9E+09,9E+09,9E+09,9E+09,9E+09]];
    VAR robtarget FillFromMoving_AbovePippet := [[-179.9398,-464.0701,468.0019],[0.004516494,-0.6988453,-6.687091E-05,0.7152586],[0,3,2,4],[-104.8699,9E+09,9E+09,9E+09,9E+09,9E+09]];
    VAR robtarget FillFromMoving3 := [[-179.954,-464.0799,435.2655],[0.004475192,-0.698854,-3.349857E-05,0.7152503],[0,3,2,4],[-104.8597,9E+09,9E+09,9E+09,9E+09,9E+09]];
    VAR robtarget FillFromMoving4 := [[-179.6848,-466.2216,337.4254],[0.01326209,0.01003572,0.7071167,-0.7069012],[0,2,1,4],[-137.6343,9E+09,9E+09,9E+09,9E+09,9E+09]];
    VAR robtarget FillFromMoving5 := [[-179.6848,-466.2216,337.4254],[0.01326209,0.01003572,0.7071167,-0.7069012],[0,2,1,4],[-137.6343,9E+09,9E+09,9E+09,9E+09,9E+09]];
    VAR robtarget FillFromMoving6 := [[-179.6848,-466.2216,337.4254],[0.01326209,0.01003572,0.7071167,-0.7069012],[0,2,1,4],[-137.6343,9E+09,9E+09,9E+09,9E+09,9E+09]];
    CONST robtarget cap1 :=[[539.2289,-80.78963,155.071],[0.0006984808,-0.09972568,0.9949208,-0.01366684],[0,-1,0,0],[113.2584,9E+09,9E+09,9E+09,9E+09,9E+09]];
    CONST robtarget cap2 :=[[539.3752,-80.91126,149.634],[0.0111098,0.7141981,0.6998098,-0.007997087],[0,-1,1,0],[113.2606,9E+09,9E+09,9E+09,9E+09,9E+09]];
    CONST robtarget cap3 :=[[539.2651,-80.9881,156.9109],[0.01106579,0.7123331,0.7017086,-0.0080128],[0,-1,1,0],[113.2854,9E+09,9E+09,9E+09,9E+09,9E+09]];


    VAR robtarget RemoveMovingWeirdJar1 := [[269.7121,-585.5166,233.3951],[0.05361825,-0.8542708,-0.5169712,0.009342714],[0,-1,1,4],[153.0393,9E+09,9E+09,9E+09,9E+09,9E+09]];
    VAR robtarget RemoveMovingWeirdJar2 := [[262.6859,-605.2153,70.33295],[0.02038794,0.8365789,0.545913,-0.04121916],[1,-1,1,4],[-156.4207,9E+09,9E+09,9E+09,9E+09,9E+09]];
    VAR robtarget RemoveStationaryWeirdJar2 := [[336.9096,-587.9133,67.63241],[0.001629263,0.8629555,0.5051923,0.009270674],[1,-1,1,4],[-161.3788,9E+09,9E+09,9E+09,9E+09,9E+09]];

    CONST robtarget ClampBase:= [[-19.13844,-434.3788,73.91506],[0.008910468,-0.03634905,-0.9992893,0.004494478],[0,-1,-1,4],[-122.7832,9E+09,9E+09,9E+09,9E+09,9E+09]];
    CONST robtarget ClampSet:= [[-124.8309,-491.0456,124.9815],[0.009361908,0.7046296,-0.7095054,-0.003409618],[0,0,-2,4],[-115.1052,9E+09,9E+09,9E+09,9E+09,9E+09]];
    var robtarget ClampVar;
    var robtarget ClampVar2;



ENDMODULE
